{attribute 'GeneratedUsingTerminal: EL3773-0000-0016'}
{attribute addProperty BoxType "EL3773-0000-0016"}
{attribute addProperty Id "Cycle_CountAT %I*UINT2"}
{attribute addProperty CRC "2980656546"}
{attribute addProperty Size "2"}
TYPE AI_CycleCount_B1A935A2 EXTENDS InputBase_8311D824 :
STRUCT
	{attribute addProperty Name "Cycle_Count"}
	Cycle_Count AT %I* : UINT;
END_STRUCT
END_TYPE

(* stored: Version 1.2.0.0, ProductVersion 3.1.4024.11
   DUT AI_CycleCount_B1A935A2: Id {850c76e9-bafb-4bda-ab76-1d35b7dcece3} *)
